FUNCTION_BLOCK FB_BeckhoffTaster
VAR_INPUT
	schaltend:BOOL; //true, schaltende funktion, false tastende
	Lock:BOOL:=FALSE; //Lock Input
	long_time: TIME;
END_VAR
VAR_OUTPUT
	state:BOOL:=FALSE;
END_VAR
VAR
	KeyBit AT %I*:BIT;
	LED AT %Q*:BIT;
	NotLED AT %Q*:BIT;
	KEY:BOOL;
	KeyTrig:F_TRIG;
	Key_bool_old:bool;
	keywaspushed:BOOL;
	longon:TON;
	keywaslong: BOOL;
	rising_edge: BOOL;
	falling_edge: BOOL;
END_VAR

IF KeyBit=1 THEN KEY:=TRUE; ELSE KEY:=FALSE; END_IF
IF Lock THEN 
	KEY:=FALSE;
END_IF
IF state THEN
	LED:=1;
	NotLED:=0;
ELSE
	LED:=0;
	NotLED:=1;
END_IF

IF KEY AND NOT key_bool_old THEN rising_edge:=TRUE; END_IF
IF NOT KEY AND key_bool_old THEN falling_edge:=TRUE; END_IF
IF rising_edge AND falling_edge THEN
	keywaspushed:=TRUE;
	rising_edge:=FALSE;
	falling_edge:=FALSE;
	IF schaltend THEN
		state:=NOT state;
	END_IF
END_IF

IF NOT rising_edge AND falling_edge THEN falling_edge:=FALSE; END_IF;

IF NOT schaltend THEN state:=KEY; END_IF

IF long_time > T#0S THEN
	longon(IN:=KEY,PT:=long_time);
	IF longon.Q THEN
		rising_edge:=false;
		longon.IN:=FALSE;
		keywaslong:=TRUE;
		longon();
	END_IF
END_IF
KEY_bool_old:=KEY;

METHOD isActive : BOOL
VAR_INPUT
END_VAR
isActive:=state;
END_METHOD

METHOD setOFF : BOOL
VAR_INPUT
END_VAR
state:=false;
END_METHOD

METHOD setON : BOOL
VAR_INPUT
END_VAR
state:=TRUE;
keywaspushed:=true;
END_METHOD

METHOD wasLongInput : BOOL
VAR_INPUT
END_VAR
IF keywaslong THEN
	wasLongInput:=TRUE;
	keywaslong:=FALSE;
ELSE
	wasLongInput:=false;
END_IF
END_METHOD

METHOD wasRising : BOOL
VAR_INPUT
END_VAR
wasRising:=keywaspushed;
keywaspushed:=false;
END_METHOD

END_FUNCTION_BLOCK

(* stored: Version 1.1.0.1, ProductVersion 3.1.4022.9
   POU FB_BeckhoffTaster: Id {e6bb3d27-afda-40cb-bb1b-b1fb22b38c68}, SpecialFunc None
   Method isActive: Id {4ee469b8-93f8-4ce2-b77a-81d4b84e0d2d}
   Method setOFF: Id {950ef05b-d402-4eb1-adaa-ceefeee4b6d0}
   Method setON: Id {51331d44-f28e-4357-a38b-36c6cffeb542}
   Method wasLongInput: Id {1a5d00d2-86c6-46b9-b81a-5af9c49c0ac8}
   Method wasRising: Id {5518e2c2-3075-44f1-8c32-26091beeff42} *)
